// TIA Portal V18 export
DATA_BLOCK "BO_Torq_DB"   // DB33
// stored: AutoNumber false, InstanceOfName BO_Torq, InstanceOfType FB
"BO_Torq"
   // VAR_INPUT
   //    Start : Bool;
   // END_VAR
   // VAR_OUTPUT
   //    FlowRevmAOut : Real;
   //    EnableP1 : Bool;
   //    EnableP2 { ExternalWritable := 'False'} : Bool;
   //    BOEn : Bool;
   //    BOSeqRunning : Bool;
   // END_VAR
   // VAR
   //    PumpToggle : Bool;
   //    RampDown : Bool;
   //    RampDownComplete : Bool;
   //    Flow_Ramp { S7_SetPoint := 'True'} : RampFunction;
   //    FlowRampInmA : Real;
   //    BOFlowmA : Real;
   //    BOSeqRunLast : Bool;
   // END_VAR
BEGIN
END_DATA_BLOCK
